Staubli VAL3: findTrajItem.pgx

program findTrajItem(InstrItem x_iItem, num& x_nResult)
  local num i
  local string l_sPath
  local num l_nSize
  local num j
  local string l_sItem
  local num l_nSizeItem
  local num k
  local TrajectoryItem l_tTraj
  local num z
  local bool l_bnFound
  local string l_sMessage
  local string l_sSession
  local num l_nResult
  local bool l_bFound
begin
  // scan all the trajectory
  for i=0 to size(saveData:sTrajType)-1
    call saveData:getPathInstr(saveData:sTrajType[i],l_sPath)
    // TRAJECTORY
    l_nResult=TrajItem:libLoad(l_sPath)
    delay(0)
    if l_nResult==0
      call TrajItem:getSize(l_nSize)
      for j=0 to l_nSize-1
        // load the trajectory
        call TrajItem:get(l_sItem,j)
        call saveData:getSession(l_sSession)
        // SHOW THE trajectory name
        l_sMessage="SESSION:"+l_sSession+">"+saveData:sTrajType[i]+" "+l_sItem
        call use:typeLen(1,5,l_sMessage,38)
        call TrajItem:load(l_sItem,x_nResult)
        if x_nResult==0
          call TrajItem:getSizeItem(false,l_nSizeItem)
          // scan for the action
          for k=0 to l_nSizeItem-1
            // get the item
            call TrajItem:getTrajItem(l_tTraj,k)
            // scan deeper for all the action
            for z=0 to size(l_tTraj.iInstr)-1
              // look inside
              l_bFound=(l_tTraj.iInstr[z].sType==x_iItem.sType and(l_tTraj.iInstr[z].sData==x_iItem.sData or find(l_tTraj.iInstr[z].sData,x_iItem.sData+">")!=-1))
              // use nested items
              l_bFound=l_bFound or find(l_tTraj.iInstr[z].sType+" "+l_tTraj.iInstr[z].sData,x_iItem.sData)!=-1
              // FOUND IT
              if l_bFound
                x_nResult=-1
                call language:message(l_sMessage,23)
                popUpMsg(l_sMessage+x_iItem.sType+" "+x_iItem.sData+chr(10)+"SESSION:"+l_sSession+chr(10)+saveData:sTrajType[i]+" "+l_sItem+" > "+l_tTraj.iInstr[z].sType+" "+l_tTraj.iInstr[z].sData)
                // back
                return
              endIf
            endFor
          endFor
        else
          popUpMsg("error loading...SESSION:"+l_sSession+">"+saveData:sTrajType[i]+" "+l_sItem+" error "+toString("",x_nResult))
        endIf
      endFor
    endIf
  endFor
end
